(* PLC project clamping, Dassault Systèmes ControlBuild 2024x *)
(* stored: creationDateTime 2023-10-03T11:13:44-01:00 *)

FUNCTION_BLOCK drill.clamping
  VAR_INPUT
    acknowledgePB : BOOL := false;
  END_VAR
  VAR_INPUT
    releasing : BOOL := false;
    clamping : BOOL := false;
  END_VAR
  VAR_INPUT
    rightUnlocked : BOOL := false;
    rightLocked : BOOL := false;
  END_VAR
  VAR_INPUT
    leftUnlocked : BOOL := false;
    leftLocked : BOOL := false;
  END_VAR
  VAR_INPUT
    rightFault : BOOL := false;
    leftFault : BOOL := false;
  END_VAR
  VAR_OUTPUT
    clampingOK : BOOL := false;
    releasingOK : BOOL := false;
    clampingFault : DINT := 0;
  END_VAR
  VAR_OUTPUT
    rightLocking : BOOL := false;
  END_VAR
  VAR_OUTPUT
    leftLocking : BOOL := false;
  END_VAR
  VAR CONSTANT
    clampingDuration : DINT := 110;
    releasingDuration : DINT := 110;
  END_VAR

INITIAL_STEP 10:
  10_INLINE1(N);
  COMPUTE_FUNCTION_BLOCKS(S);
END_STEP
ACTION 10_INLINE1:
  IF (clampingFault = 0) THEN
  	releasingOK;
  END_IF;
END_ACTION
TRANSITION FROM 10 TO 11
  := clamping AND NOT releasing AND (clampingFault = 0);
END_TRANSITION
STEP 11:
END_STEP
TRANSITION FROM 11 TO 12
  := rightLocked AND leftLocked;
END_TRANSITION
TRANSITION FROM 11 TO 13
  := releasing AND NOT clamping;
END_TRANSITION
TRANSITION FROM 11 TO 14
  := (clampingFault > 0);
END_TRANSITION
STEP 12:
  12_INLINE2(N);
END_STEP
ACTION 12_INLINE2:
  clampingOK;
END_ACTION
TRANSITION FROM 12 TO 13
  := releasing AND NOT clamping AND (clampingFault = 0);
END_TRANSITION
STEP 13:
END_STEP
TRANSITION FROM 13 TO 10
  := rightUnlocked AND leftUnlocked;
END_TRANSITION
TRANSITION FROM 13 TO 11
  := clamping AND NOT releasing;
END_TRANSITION
TRANSITION FROM 13 TO 14
  := (clampingFault > 0);
END_TRANSITION
STEP 14:
END_STEP
TRANSITION FROM 14 TO 10
  := rightUnlocked AND leftUnlocked;
END_TRANSITION
ACTION COMPUTE_FUNCTION_BLOCKS:  (* blocks drawn on the SFC sheet *)
  G1:
END_ACTION

ACTION PreSFC:
IF(((X10 OR X12) AND RE acknowledgePB )) THEN
	clampingFault := 0;
END_IF;
IF(X11 AND rightFault) THEN
	clampingFault := 1;
END_IF;
IF(X11 AND leftFault) THEN
	clampingFault := 2;
END_IF;
IF(X13 AND rightFault) THEN
	clampingFault := 3;
END_IF;
IF(X13 AND leftFault) THEN
	clampingFault := 4;
END_IF;
END_ACTION

ACTION PostSFC:
leftLocking := X11 OR X12;
rightLocking := X11 OR X12;
END_ACTION
END_FUNCTION_BLOCK
